FUNCTION_BLOCK FB_VolumeFlow_EL3054 IMPLEMENTS I_VolumeFlowSensor
VAR_INPUT
END_VAR
VAR_OUTPUT
END_VAR
VAR
	//Property Real value
	fVolFlow : REAL;
	//Raw value
	VolFlowRaw AT %I* : INT;
	//Convertion parameters
	m : REAL := 0.000366222026; //Multiplier for convertion
END_VAR

PROPERTY VolumeFlow : REAL
GET
fVolFlow := m * INT_TO_REAL(VolFlowRaw);
VolumeFlow := THIS^.fVolFlow;
END_GET
END_PROPERTY

END_FUNCTION_BLOCK

(* stored: Version 1.1.0.1
   POU FB_VolumeFlow_EL3054: Id {0c1f86b8-d855-4a32-ba8b-f5b6e88ec322}, SpecialFunc None
   Property VolumeFlow: Id {a420b916-67af-406a-bbd1-8413364e2f5d}
   Get Get: Id {19e69505-7e17-4d06-a20f-c5112e8c91f5} *)
